// TIA Portal V18 export
TYPE "LGasp_typeHMI_zona"
// stored: IsFailsafeCompliant false
   STRUCT
      abilitata : Bool;   // 1 = zona presente nella linea
      nome : WString[20];
      AUTOman : Bool;   // 0=manuale 1=automatico
      MARCIAstop : Bool;   // 1=marcia
      allarmi : Bool;   // allarmi presenti in sezione
      warning : Bool;   // warning presenti in sezione
      fungointervenuto : Bool;   // fungo intervenuto per 10'
      cancellointervenuto : Bool;   // cancello intervenuto per 10'
      barrieraintervenuta : Bool;   // barriera intervenuta per 10'
      safetydevice : Array[1.."N_SAFETYDEVICE"] of "LGasp_typeHMI_safetydevice";   // dispositivi di sicurezza
   END_STRUCT;
END_TYPE
